// TIA Portal V20 export
DATA_BLOCK "DB_ConveyorParameters"   // DB25
// stored: Access Published, MemoryReserve 100, Namespace LineC1
   VAR
      Line : Struct
         C1 : Struct
            Conveyor : Array[_.minC1.._.maxC1] of "Global.ConveyorParameters";
            MABS { S7_SetPoint := 'True'} : Array[_."MABS_C1.2.1".._."MABS_C1.2.2"] of "Global.MABS_Setpoint";
            Transfer : Array[_."Transfer_C1.13.1".._."Transfer_C1.14.1"] of "LineC1.setTransferTimer";
         END_STRUCT;
      END_STRUCT;
   END_VAR
BEGIN
END_DATA_BLOCK
